// Mitsubishi GX Works2 project: ServMotor   PLC: Q03UDV

PROGRAM MAIN
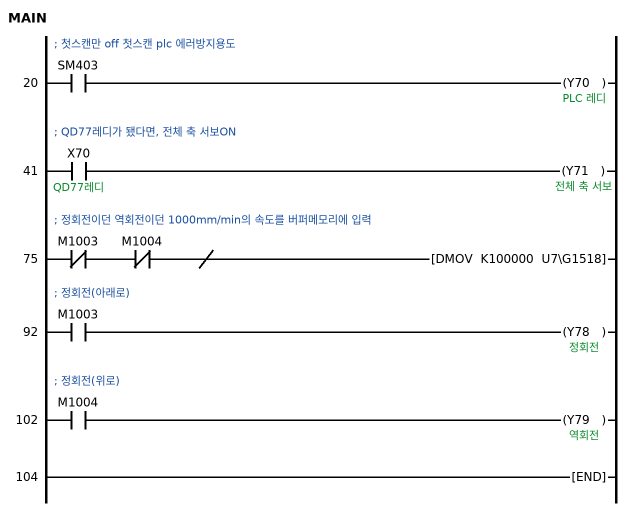
; 첫스캔만 off 첫스캔 plc 에러방지용도
20    LD      SM403
      OUT     Y70  ; PLC 레디
; QD77레디가 됐다면, 전체 축 서보ON
41    LD      X70  ; QD77레디
      OUT     Y71  ; 전체 축 서보
; 정회전이던 역회전이던 1000mm/min의 속도를 버퍼메모리에 입력
75    LDI     M1003
      ANI     M1004
      INV
      DMOV    K100000 U7\G1518
; 정회전(아래로)
92    LD      M1003
      OUT     Y78  ; 정회전
; 정회전(위로)
102   LD      M1004
      OUT     Y79  ; 역회전
104   END
END_PROGRAM
